FUNCTION_BLOCK Ass_Pallet
VAR_INPUT
END_VAR
VAR_OUTPUT
END_VAR
VAR
END_VAR

END_FUNCTION_BLOCK

(* stored: Version 1.1.0.1, ProductVersion 3.1.4024.16
   POU Ass_Pallet: Id {07db0394-8679-47b5-a6db-93ce50ed8062}, SpecialFunc None *)
